FUNCTION WRITE_PROTECTED_WORD
VAR_INPUT
    Ptr : POINTER TO WORD;
    Value : WORD;
END_VAR

Ptr^ := Value;

END_FUNCTION

(* stored: Version 1.1.0.1, ProductVersion 3.1.4022.18
   POU WRITE_PROTECTED_WORD: Id {00031d54-f0f1-405a-8c1e-ac2fc1af74f9}, SpecialFunc None *)
